(* Schneider Machine Expert - Basic project Industrial_Zone_192_168_10_72, file version 1.8.0.0 *)
(* ProjectInformations: Name=New project *)

HARDWARE
  Cpu 0: TM221CE16R
  EthernetConfiguration: NetworkName=M221, IpAllocationMode=FixedAddress, IpAddress=172.18.212.88, SubnetMask=255.255.255.0
  SerialLineConfiguration: Baud=Baud19200, Parity=ParityEven, DataBits=DataBits8, StopBits=StopBits1, PhysicalMedium=PhysicalMediumRs485, TransmissionMode=TransmissionModeModbusRtu, SlaveId=1, Addressing=SlaveAddressing
  MastTask: UsePeriodScanMode=false, PeriodScan=100
  FastTask: Period=255
  CpuBehavior: StartingMode=StartAsPreviousState, AutoSaveRamOnEeprom=true, WatchdogPeriod=250

SYMBOLS  (address, symbol, comment, settings)
  %M30        "Attack Bit"
  %M40        "Attack Enable Bit"
  %TM0        [Type=TOF, Preset=25, Base=OneSecond]
  %Q0.0       "Runway Leds"
  %Q0.1       "Power Plant"
  %Q0.2       "Pylon LEDs"
  %Q0.3       "Runway LEDs"
  %Q0.5       "Red Light"
  %Q0.6       "White Light"

POU New POU
  (* SectionNumber=1 *)

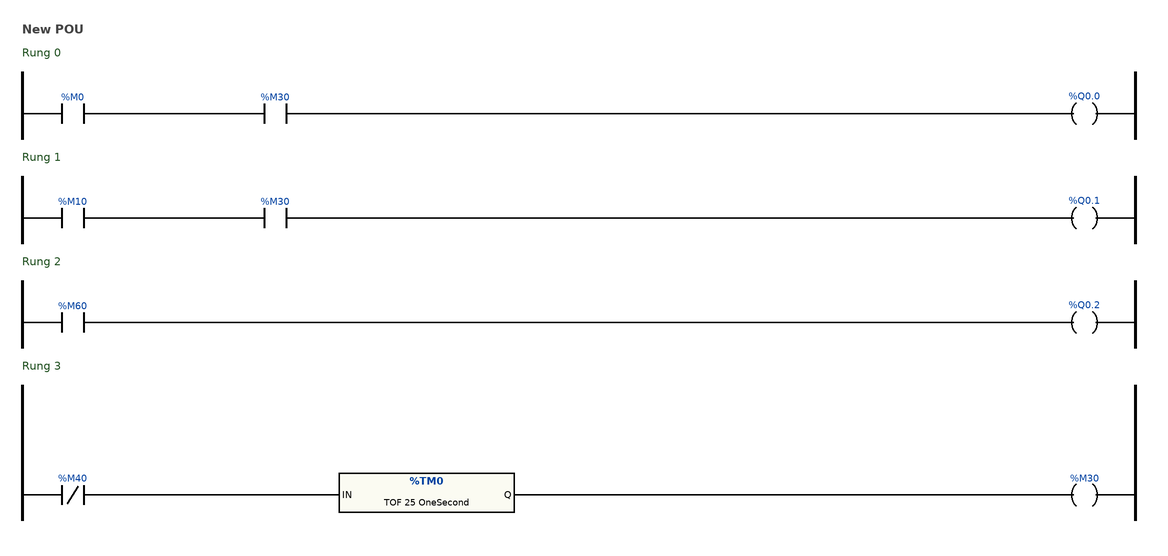

// Rung 0
  LD %M0
  AND %M30
  ST %Q0.0
  // as ST:
  //   %Q0.0 := %M0 AND %M30;

// Rung 1
  LD %M10
  AND %M30
  ST %Q0.1
  // as ST:
  //   %Q0.1 := %M10 AND %M30;

// Rung 2
  LD %M60
  ST %Q0.2
  // as ST:
  //   %Q0.2 := %M60;

// Rung 3
  BLK %TM0
  LDN %M40
  IN
  OUT_BLK
  LD Q
  ST %M30
  END_BLK
  // as ST:
  //   %TM0(IN := NOT %M40);
  //   %M30 := %TM0.Q;
